{attribute 'pack_mode' := '1'}
TYPE TRunDataPearling :
STRUCT
		abUseSpindle				: ARRAY[0..1] OF BOOL;
		sPearlingData				: TPearlingDataHead;
		iLayringPos					: INT;
		iLayringOffsetPos				: INT;
		apsPartData					: ARRAY[0..1] OF POINTER TO TPartData;
		bForceSharpenAfterPearling	: BOOL;
END_STRUCT
END_TYPE

(* stored: Version 1.1.0.1, ProductVersion 3.1.4022.12
   DUT TRunDataPearling: Id {2c0a72c0-fe81-4d5c-a494-76b0cd46f827} *)
